{attribute 'pack_mode' := '1'}
TYPE ST_StopMotion EXTENDS ST_MsgToPLC:
STRUCT
    
END_STRUCT
END_TYPE

(* stored: Version 1.1.0.1, ProductVersion 3.1.4022.18
   DUT ST_StopMotion: Id {8c3aaf65-03ea-4971-8c90-c684b5fd56a6} *)
